PROGRAM MAIN
VAR
	ServoDo:BOOL;
	ServoDone: BOOL;
	ServoAngle:REAL;
	CurrentAngle:REAL;
	FixtureEnable:BOOL;
	Controller:ServoControl;
	//Spray block
	spray:Spray;
	SprayExecute:BOOL:=TRUE;
	
	Order:ARRAY[0..7] OF INT:=[1,2,3,4,5,6,7,8];
	//get spin before servo step to get 1 at head
	FixtureState:INT:=0;
	temp:INT:=0;
	FixtureStateArray:ARRAY[0..7] OF BOOL:=[0,0,0,0,0,0,0,0];
	i: INT;
END_VAR

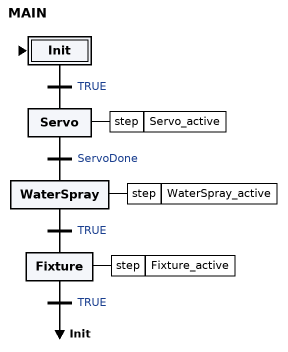
INITIAL_STEP Init:
END_STEP
TRANSITION FROM Init TO Servo
    := TRUE;
END_TRANSITION
STEP Servo:
    Servo_active(N);  // step action
END_STEP
TRANSITION FROM Servo TO WaterSpray
    := ServoDone;
END_TRANSITION
STEP WaterSpray:
    WaterSpray_active(N);  // step action
END_STEP
TRANSITION FROM WaterSpray TO Fixture
    := TRUE;
END_TRANSITION
STEP Fixture:
    Fixture_active(N);  // step action
END_STEP
TRANSITION FROM Fixture TO Init
    := TRUE;
END_TRANSITION

ACTION Fixture_active:
temp:=1;
FOR i:=0 TO 7 DO
	FixtureStateArray[i]:= INT_TO_BOOL(REAL_TO_INT(FixtureState/temp) MOD 2);
	temp:=temp*2;
END_FOR
END_ACTION

ACTION Servo_active:
Controller(
	bExecute:=ServoDo,
	bDone=>ServoDone,
	Order=>Order,
	CurrentAngle=>CurrentAngle
);
END_ACTION

ACTION WaterSpray_active:
spray(bExecute:=SprayExecute,
	Order:=Order,
	Angle:=CurrentAngle,
	bDone=>
);
END_ACTION

END_PROGRAM

(* stored: Version 1.1.0.1, ProductVersion 3.1.4024.12
   POU MAIN: Id {230e4d08-d873-4357-920a-2f2af910e192}, SpecialFunc None
   Action Fixture_active: Id {b5409920-1ef0-47a7-a6a9-f3a909362c5a}
   Action Servo_active: Id {4d3bbd18-a0aa-4a95-984c-d65122f9c816}
   Action WaterSpray_active: Id {293afa01-2139-46ea-a09a-16ab5d22120a} *)
